// TIA Portal V16 export
// export: Created 2021-10-20T18:24:25.3067341Z, ExportSetting WithDefaults, DisplayName Totally Integrated Automation Portal, DisplayVersion V16, DisplayName TIA Portal Version Control Interface, DisplayVersion V16, DisplayName TIA Portal Openness, DisplayVersion V16, DisplayName SINAMICS Startdrive Advanced, DisplayVersion V16, DisplayName SINAMICS Startdrive G130, G150, S120, S150, SINAMICS MV, S210, DisplayVersion V16, DisplayName SINAMICS Startdrive G110M, G120, G120C, G120D, G120P, DisplayVersion V16, DisplayName STEP 7 Professional, DisplayVersion V16, DisplayName STEP 7 Safety, DisplayVersion V16, DisplayName WinCC Advanced, DisplayVersion V16
FUNCTION "Analog Alarm" : Void   // FC20, LAD
TITLE = Analog Alarm Block
VERSION : 0.1
// Checks PV against Hi_Limit and Lo_Limit alarm values
// stored: AutoNumber false, IsIECCheckEnabled false, UDAEnableTagReadback false
   VAR_INPUT
      PV : Real;   // Process Value output from PID Loop
      Hi_Limit : Real;   // Hi Alarm Value
      Lo_Limit : Real;   // Lo Alarm Value
   END_VAR
   VAR_OUTPUT
      Hi_Alarm : Bool;   // PV is in High Alarm
      Lo_Alarm : Bool;   // PV is in Low Alarm
   END_VAR
BEGIN

REGION Network 1
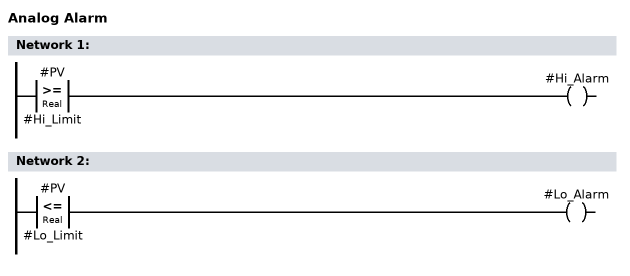
   RUNG wire#powerrail
      { S7_Templates := "SrcType := Real" } GE_Contact(in1 := #PV, in2 := #Hi_Limit)
      Coil( #Hi_Alarm )
   END_RUNG
   // the same network as SCL:
   #Hi_Alarm := #PV >= #Hi_Limit;
END_REGION

REGION Network 2
   RUNG wire#powerrail
      { S7_Templates := "SrcType := Real" } LE_Contact(in1 := #PV, in2 := #Lo_Limit)
      Coil( #Lo_Alarm )
   END_RUNG
   // the same network as SCL:
   #Lo_Alarm := #PV <= #Lo_Limit;
END_REGION
END_FUNCTION
